// TIA Portal V19 export
FUNCTION_BLOCK "MovingLight"   // FB16, SCL
TITLE = MovingLight
{ S7_Optimized_Access := 'TRUE' }
AUTHOR : Siemens
// Moving light BeltLift
// stored: IsIECCheckEnabled true, MemoryReserve 100, SetENOAutomatically true
   VAR_INPUT
      lightDirection { ExternalAccessible := 'False'; ExternalVisible := 'False'; ExternalWritable := 'False'} : Int;
      nBitsLight { ExternalAccessible := 'False'; ExternalVisible := 'False'; ExternalWritable := 'False'} : UInt;
      delay { ExternalAccessible := 'False'; ExternalVisible := 'False'; ExternalWritable := 'False'} : Time := T#200MS;   // Time delay for signal change
   END_VAR
   VAR_OUTPUT
      wrd1 { ExternalAccessible := 'False'; ExternalVisible := 'False'; ExternalWritable := 'False'} : Word;
   END_VAR
   VAR
      statDelayInt { ExternalAccessible := 'False'; ExternalVisible := 'False'; ExternalWritable := 'False'; S7_SetPoint := 'True'} : TOF_TIME;
      statGo { ExternalAccessible := 'False'; ExternalVisible := 'False'; ExternalWritable := 'False'} : Bool;
      statRun { ExternalAccessible := 'False'; ExternalVisible := 'False'; ExternalWritable := 'False'} : Time;
      statUp { ExternalAccessible := 'False'; ExternalVisible := 'False'; ExternalWritable := 'False'} : Word := 1;
      statMovingLight { ExternalAccessible := 'False'; ExternalVisible := 'False'; ExternalWritable := 'False'} : Word;
      statMaxMoveLightValue { ExternalAccessible := 'False'; ExternalVisible := 'False'; ExternalWritable := 'False'} : Word;
   END_VAR
   VAR CONSTANT
      STOP : Int;
      LEFT : Int := 10;
      RIGHT : Int := 20;
   END_VAR
BEGIN
   // function block for moving light with light direction left or right

   // calculate compare value dependent from number of LEDs used
   #statMaxMoveLightValue := 1;
   #statMaxMoveLightValue := SHL(IN := #statMaxMoveLightValue, N := (#nBitsLight - 1));

   // time delay
   #statDelayInt(IN := #statGo,
              PT := #delay,
              ET => #statRun);
   #statGo := NOT #statDelayInt.Q; // erneuter Start, wenn die Zeit abgelaufen ist


   CASE #lightDirection OF // Lauflichttypen auswählen
     #STOP:// no moving light
       #statUp := 0;

     #LEFT: // moving light left
       IF #statGo THEN
         #statMovingLight := SHR(IN := #statMovingLight, N := 1);

         IF (#statMovingLight = 0) THEN
           // set moving light to calculated value
           #statMovingLight := #statMaxMoveLightValue;
         END_IF;
         // change bytes
         // #up := SWAP(IN := #MovingLight); // SWAP only, if QW on output
         #statUp := #statMovingLight;
       END_IF;

     #RIGHT: // moving light right 
       IF #statGo THEN
         #statMovingLight := SHL(IN := #statMovingLight, N := 1);

         IF (#statMovingLight = 0) OR (#statMovingLight > #statMaxMoveLightValue) THEN
           // set first LED of moving light
           #statMovingLight := 1;
         END_IF;
         // change bytes
         // #up := SWAP(IN := #MovingLight); // SWAP only, if QW on output
         #statUp := #statMovingLight;
       END_IF;
     ELSE
       #statUp := 0;
   END_CASE;

   // output
   #wrd1 := #statUp;
END_FUNCTION_BLOCK
